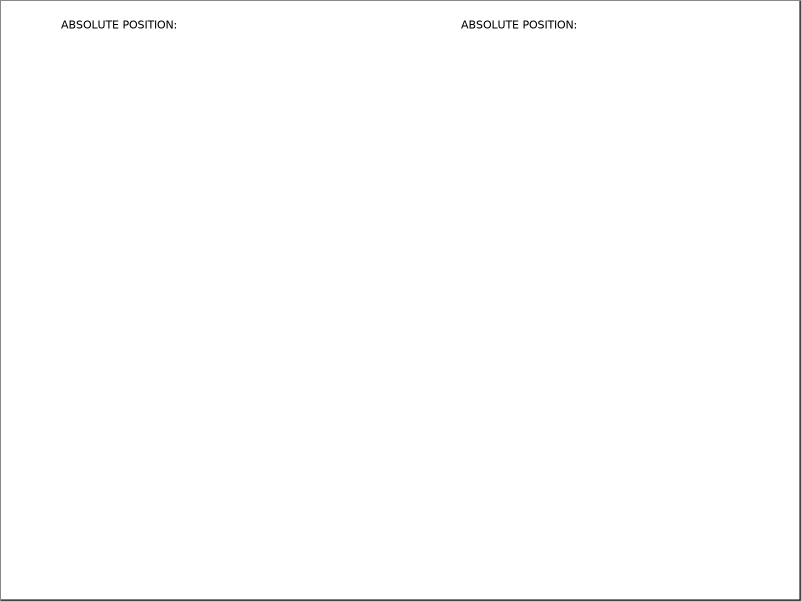
VISUALIZATION F53_Cam_Remove  // 802x602
    Rectangle (0,0 800x600)
    Label (10,10 170x30), "ABSOLUTE POSITION:"
    Label (410,10 170x30), "ABSOLUTE POSITION:"
END_VISUALIZATION

(* stored: Version 1.1.0.1, ProductVersion 3.1.4022.7
   Visu F53_Cam_Remove: Id {926bc3ea-54aa-4e84-973c-7cbae8b9057e} *)
